RoboDK station: RB ABB.rdk

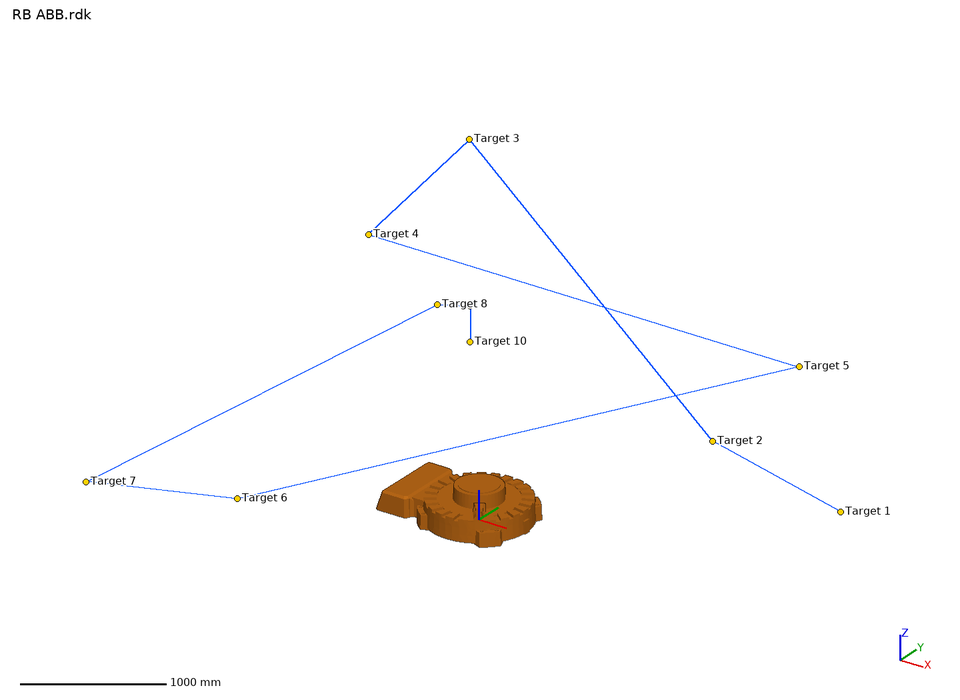
[picture v0: the station drawn from its stored meshes, robots at their saved joint values, targets as dots, program paths as lines]
Station New Station (1.1) (saved by RoboDK 5.5.4). Poses are relative to the parent item; angles as X-Y-Z fixed-axis rotations.
  - frame ABB IRB 6400 2.8 120 Base at (0, 0, 0) mm
    - robot ABB IRB 6400 2.8 120: 6 axes, payload 120 kg, reach 2800 mm, repeatability 0.1 mm, weight 2230 kg
        joint limits [-180, -70, -28, -300, -120, -300] to [180, 70, 35, 300, 120, 300]; home [0, 0, 0, 0, 0, 0]; saved at [-64.359, -30.499, -4.916, 87.645, 64.46, -84.55]
    - target Target 1 (joint target) at (2250, 1100, 250) mm, rotated rx 0 ry 90 rz 0 deg; joints [28.217, 52.944, 50.967, -145.364, 56.295, 159.027] of ABB IRB 6400 2.8 120
    - target Target 2 (joint target) at (900, 1500, 250) mm, rotated rx 0 ry 90 rz 0 deg; joints [64.983, 29.357, 65.941, -113.08, 80.073, 157.973] of ABB IRB 6400 2.8 120
    - target Target 3 (joint target) at (-850, 1100, 2220) mm, rotated rx 180 ry 0 rz -180 deg; joints [127.694, -24.532, -15.222, 180, -105.222, -52.306] of ABB IRB 6400 2.8 120
    - target Target 4 (joint target) at (-1800, 1250, 1170) mm, rotated rx -180 ry 0 rz 180 deg; joints [145.222, 15.964, 22.324, 0, 67.676, 145.222] of ABB IRB 6400 2.8 120
    - target Target 5 (joint target) at (1800, 1250, 1170) mm, rotated rx 0 ry 90 rz 0 deg; joints [37.999, 11.115, 30.096, -122.695, 47.016, 133.272] of ABB IRB 6400 2.8 120
    - target Target 6 (joint target) at (-1250, -1100, 250) mm, rotated rx 0 ry 90 rz 0 deg; joints [-142.815, 34.776, 62.733, -139.521, -111.408, 17.302] of ABB IRB 6400 2.8 120
    - target Target 7 (joint target) at (-2250, -1480, 250) mm, rotated rx 180 ry 0 rz -180 deg; joints [-146.664, 63.554, 35.904, 0, 54.096, -146.664] of ABB IRB 6400 2.8 120
    - target Target 8 (joint target) at (450, -1140, 2220) mm, rotated rx 0 ry 90 rz 0 deg; joints [-77.631, -40.204, -13.545, 87.06, 77.98, -76.145] of ABB IRB 6400 2.8 120
    - target Target 9 (joint target) at (800, -1250, 2350) mm, rotated rx 0 ry 90 rz 0 deg; joints [-64.359, -26.13, -13.162, 83.763, 65.079, -75.459] of ABB IRB 6400 2.8 120
    - target Target 10 (joint target) at (800, -1250, 2075) mm, rotated rx 0 ry 90 rz 0 deg; joints [-64.359, -30.499, -4.916, 87.645, 64.46, -84.55] of ABB IRB 6400 2.8 120
  - program Prog1 (11 instructions, listed below)
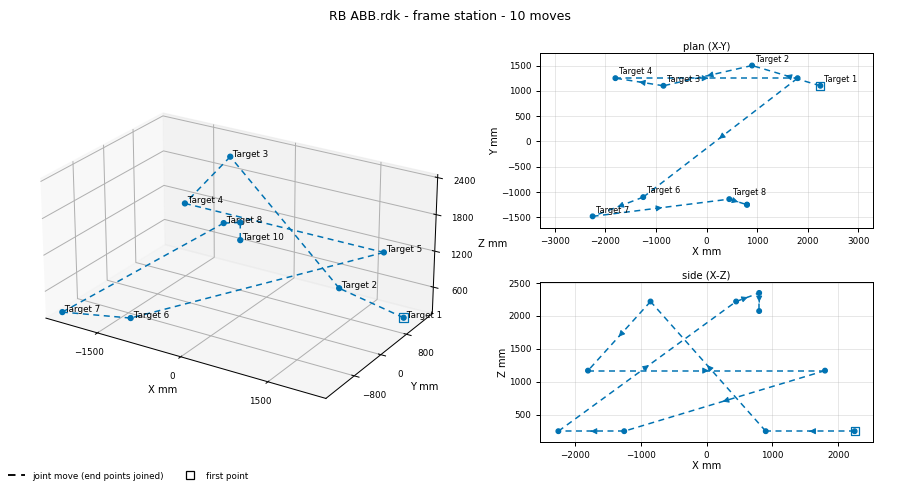
[picture p0: tool path of RB ABB.rdk in frame station, 10 of 10 moves have a stored position in this frame; points joined in program order, loops and branches not executed]

--- program Prog1 (robot ABB IRB 6400 2.8 120) ---
  Set Ref.: ABB IRB 6400 2.8 120 Base
  MoveJ (Target 1)
  MoveJ (Target 2)
  MoveJ (Target 3)
  MoveJ (Target 4)
  MoveJ (Target 5)
  MoveJ (Target 6)
  MoveJ (Target 7)
  MoveJ (Target 8)
  MoveJ (Target 9)
  MoveJ (Target 10)
